TYPE MNG_APPLICATION_OUTPUTS_32BIT :
STRUCT
    NumSignals                     : INT     := 0         ;
END_STRUCT
END_TYPE

(* stored: Version 1.1.0.1, ProductVersion 3.1.0.23
   DUT MNG_APPLICATION_OUTPUTS_32BIT: Id {e82eddb4-48f9-45b7-ac63-6d2a52490074} *)
